// Mitsubishi GX Works2 project: fk2n_test_in_out   PLC: FX2N/FX2NC

PROGRAM MAIN
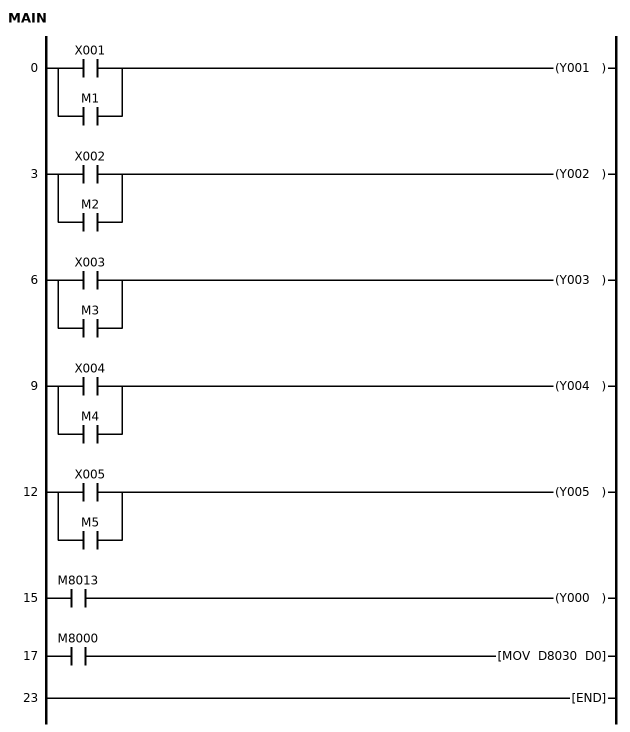
0     LD      X001
      OR      M1
      OUT     Y001
3     LD      X002
      OR      M2
      OUT     Y002
6     LD      X003
      OR      M3
      OUT     Y003
9     LD      X004
      OR      M4
      OUT     Y004
12    LD      X005
      OR      M5
      OUT     Y005
15    LD      M8013
      OUT     Y000
17    LD      M8000
      MOV     D8030 D0
23    END
END_PROGRAM
